{attribute 'linkalways'} 
{attribute 'no_explicit_call' := 'This FB is a CLASS and must be accessed using methods or properties'}
{attribute 'enable_dynamic_creation'}
FUNCTION_BLOCK Node_F_VN_CopyIntoDisplayableImage EXTENDS VisionNode
VAR
    ipSrcImage : _ITcVnImage;
    ipDestImage : _ITcVnDisplayableImage;
    hrPrev : _HRESULT(S_OK);
	hresult : _HRESULT(S_OK);
END_VAR

METHOD PUBLIC  Clone : I_Node
VAR
	pNode : POINTER TO Node_F_VN_CopyIntoDisplayableImage;
END_VAR
pNode := __NEW(Node_F_VN_CopyIntoDisplayableImage);
Clone := pNode^;
END_METHOD

METHOD FB_init : BOOL
VAR_INPUT
	bInitRetains : BOOL; // if TRUE, the retain variables are initialized (warm start / cold start)
	bInCopyCode : BOOL;  // if TRUE, the instance afterwards gets moved into the copy code (online change)
END_VAR
AddInput('ipSrcImage', ipSrcImage);
AddInput('hrPrev', hrPrev);
AddOutput('ipDestImage', ipDestImage);
AddOutput('hresult',hresult);
END_METHOD

METHOD PROTECTED OnExecute
hresult.Value := F_VN_CopyIntoDisplayableImage(
    ipSrcImage := ipSrcImage.Value,
	ipDestImage := ipDestImage.Value,
	hrPrev:= hrPrev.Value);
END_METHOD

METHOD PUBLIC PreExecutionCheck
VAR_INPUT
	Check : I_PreExecutionChecks;
END_VAR
Check.IsTrue(ipSrcImage.IsValid, 'ipSrcImage must contain an image');
END_METHOD

END_FUNCTION_BLOCK

(* stored: Version 1.1.0.1, ProductVersion 3.1.4024.15
   POU Node_F_VN_CopyIntoDisplayableImage: Id {b024eae5-a9db-0e06-2e5b-efcbe86d929d}, SpecialFunc None
   Folder Constructor: Id {b8656419-8d5d-034a-1d91-fec4b31856d9}
   Method Clone: Id {c1036455-ed8d-0b43-26fd-729cee54e744}
   Method FB_init: Id {7a3e7157-f154-071b-2aac-bd750e188bf0}
   Method OnExecute: Id {b5480678-839a-0a85-0ad3-acb6be2ceb19}
   Method PreExecutionCheck: Id {c29e4874-e3e6-0c26-2ab6-30b5f67b3b23} *)
